FUNCTION_BLOCK PUBLIC FB_AmericanPizzaNewYork EXTENDS FB_AmericanPizzaMargherita
VAR_INPUT
END_VAR
VAR_OUTPUT
END_VAR
VAR
	bBroccoli	: BOOL := TRUE;
	bMushroom	: BOOL := TRUE;
END_VAR

PROPERTY PUBLIC bHasBroccoli : BOOL
GET
bHasBroccoli := this^.bBroccoli;
END_GET
SET
this^.bBroccoli := bHasBroccoli;
END_SET
END_PROPERTY

PROPERTY PUBLIC bHasMushroom : BOOL
GET
bHasMushroom := this^.bMushroom;
END_GET
SET
this^.bMushroom := bHasMushroom;
END_SET
END_PROPERTY

METHOD PUBLIC GetPrice : LREAL
VAR_INPUT
END_VAR
GetPrice := SUPER^.GetPrice();
IF (THIS^.bBroccoli) THEN
	GetPrice := GetPrice + 0.8;
END_IF
IF (THIS^.bMushroom) THEN
	GetPrice := GetPrice + 0.75;
END_IF
END_METHOD

END_FUNCTION_BLOCK

(* stored: Version 1.1.0.1, ProductVersion 3.1.4022.12
   POU FB_AmericanPizzaNewYork: Id {ded0108f-44c4-4733-bef4-21814fff2981}, SpecialFunc None
   Property bHasBroccoli: Id {66e6f12d-88dd-4e05-a33e-94a248d60984}
   Get Get: Id {73a1929f-75e4-491b-8571-66a2a9810319}
   Set Set: Id {790dd8b0-e942-42a2-82f8-eb0b9153f3f7}
   Property bHasMushroom: Id {4f57592b-a619-4e81-9895-4261a626186c}
   Get Get: Id {38b67d32-6abe-4d34-bc92-e2edcc3b08c3}
   Set Set: Id {3657790e-1c6c-4265-9138-37441704b62b}
   Method GetPrice: Id {00705aee-2a37-4be1-8c79-d8c8214fba91} *)
